// TIA Portal V20 export
DATA_BLOCK "InstCallGlobal"   // DB265
// stored: InstanceOfName CallGlobal, InstanceOfType FB
"CallGlobal"
   // VAR
   //    statClockSysMemOld { ExternalWritable := 'False'} : Byte;
   //    statPulse : Array[0..9] of Bool;
   //    instLAF_PowerOnOff { ExternalWritable := 'False'} : "LAF_PowerOnOff";
   //    instLAF_HmiHeaderManager { ExternalWritable := 'False'} : "LAF_HmiHeaderManager";
   //    instLAF_ClockGen { ExternalWritable := 'False'} : "LAF_ClockGenerator";
   //    instLSNTP_Server { ExternalWritable := 'False'} : "LSNTP_Server";
   //    statTonTimer { ExternalWritable := 'False'} : Array[0..9] of TON_TIME;
   // END_VAR
BEGIN
END_DATA_BLOCK
